FUNCTION Convert_DT_TO_DT : Hresult
VAR_INPUT
	in : DT;
	out : REFERENCE TO DT;
END_VAR

out := in;

END_FUNCTION

(* stored: Version 1.1.0.1, ProductVersion 3.1.4024.12
   POU Convert_DT_TO_DT: Id {2cf209c1-c3f7-47c9-8ec9-ba0ad1566d33}, SpecialFunc None *)
